Staubli VAL3: default.pjx

Parameters millimeterUnit=true stackSize=5000 version=s8.3.1cs9_BS885
Program file=start.pgx
Program file=stop.pgx
Data file=default.dtx
